TYPE T_Error : ST_ERROR; END_TYPE

(* stored: Version 1.1.0.1, ProductVersion 3.1.4024.4
   DUT T_Error: Id {6e9c0c59-1542-0b98-2224-2648086575dc} *)
